{attribute 'qualified_only'}
TYPE E_ManualPrimeState :
(
    Idle := 0,
    ExtendingSupport,
    CheckingPart,
	WaitingForNozzlePressure,
    BuildingVacuum,
    StartingPrime,
    WaitingPrime,
    ReleasingVacuum,
    RetractingSupport,
    Complete,
    Aborting
);
END_TYPE

(* stored: Version 1.1.0.1, ProductVersion 3.1.4026.18
   DUT E_ManualPrimeState: Id {8be5667d-801a-438e-a326-e6bbda5039b7} *)
